// Mitsubishi GX Works2 project: mc1   PLC: FX1N/FX1NC

PROGRAM MAIN
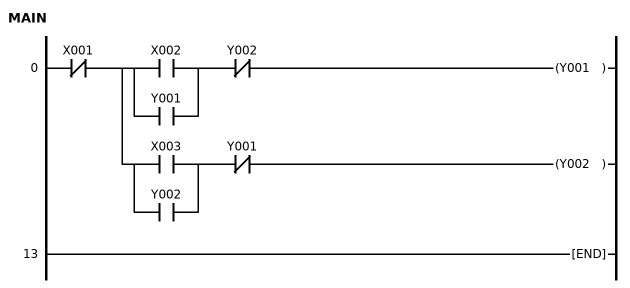
0     LDI     X001
      MPS
      LD      X002
      OR      Y001
      ANB
      ANI     Y002
      OUT     Y001
      MPP
      LD      X003
      OR      Y002
      ANB
      ANI     Y001
      OUT     Y002
13    END
END_PROGRAM
